// TIA Portal project "Tetsi" (V15.1)

(* hardware
DEVICE "S71500/ET200MP station_1"  S7-1500 station
   slot 0: "Rail_0"  Rack  6ES7 590-1***0-0AA0
   slot 1: "PLC_1"  CPU 1511-1 PN  6ES7 511-1AK02-0AB0  V2.6
      slot 3: "CPU display_1"  6ES7591-1AA00-0AA0
   slot 2: "DI 16x24VDC / DQ 16x24VDC/0.5A BA_1"  DI 16/DQ 16x24VDC  6ES7 523-1BL00-0AA0  V1.0
   slot 3: "AI/AQ 4xU/I/RTD/TC / 2xU/I ST_1"  AI/AQ 4xU/I/RTD/TC / 2xU/I ST  6ES7 534-7QE00-0AB0  V1.0
*)

// ===== PLC "PLC_1"  CPU 1511-1 PN =====

VAR_GLOBAL   // PLC tag table "Default tag table"
   "Clock_Byte" AT %MB0 : Byte;
   "Clock_10Hz" AT %M0.0 : Bool;
   "Clock_5Hz" AT %M0.1 : Bool;
   "Clock_2.5Hz" AT %M0.2 : Bool;
   "Clock_2Hz" AT %M0.3 : Bool;
   "Clock_1.25Hz" AT %M0.4 : Bool;
   "Clock_1Hz" AT %M0.5 : Bool;
   "Clock_0.625Hz" AT %M0.6 : Bool;
   "Clock_0.5Hz" AT %M0.7 : Bool;
   "Tag_1" AT %M100.0 : Bool;
   "Tag_2" AT %M100.2 : Bool;
   "Tag_3" AT %M100.3 : Bool;
   "Tag_4" AT %M100.4 : Bool;
END_VAR

VAR_GLOBAL   // PLC tag table "Tagit"
   "ColorSensor" AT %MW10 : Int;
   "ConveyorEntry" AT %Q0.0 : Bool;
   "ConveyorExit" AT %Q0.1 : Bool;
   "RotationArm" AT %Q0.2 : Bool;
   "RotationArm2" AT %Q0.3 : Bool;
   "RotationArm3" AT %Q0.4 : Bool;
   "StartButton" AT %M12.0 : Bool;
   "StopButton" AT %M12.1 : Bool;
   "ActButton" AT %M12.2 : Bool;
   "RetroreflectiveSensors" AT %M12.3 : Bool;
   "RetroreflectiveSensors2" AT %M12.4 : Bool;
   "RetroreflectiveSensors3" AT %M12.5 : Bool;
END_VAR

DATA_BLOCK "DB"   // DB1
{ S7_Optimized_Access := 'FALSE' }
VERSION : 0.1
   VAR
      nLaatikoita : Int;
      nLaatikoitaSisaan : Int;
      nLaatikoitaUlos : Int;
      kulj2_tyhjenna : Bool;
      kulj1_seis : Bool;
   END_VAR
BEGIN
END_DATA_BLOCK

DATA_BLOCK "Data_block_1"   // DB2
{ S7_Optimized_Access := 'FALSE' }
VERSION : 0.1
   VAR
      start : Bool;
      stop : Bool;
      anturi1 : Bool;
      turvakytkin : Bool;
   END_VAR
BEGIN
END_DATA_BLOCK

DATA_BLOCK "opc_test"   // DB3
{ S7_Optimized_Access := 'TRUE' }
VERSION : 0.1
   VAR
      "bool" : Bool;
      "int" : Int;
   END_VAR
BEGIN
END_DATA_BLOCK

ORGANIZATION_BLOCK "Main"   // OB1, LAD, ProgramCycle
TITLE = "Main Program Sweep (Cycle)"
{ S7_Optimized_Access := 'TRUE' }
VERSION : 0.1
   VAR_INPUT
      Initial_Call : Bool;   // Initial call of this OB
      Remanence : Bool;   // =True, if remanent data are available
   END_VAR
   VAR_TEMP   // added for the SCL form of the ladder/FBD networks
      _w1 : Bool;
      _w2 : Bool;
   END_VAR
BEGIN

REGION Network 1: start/stop
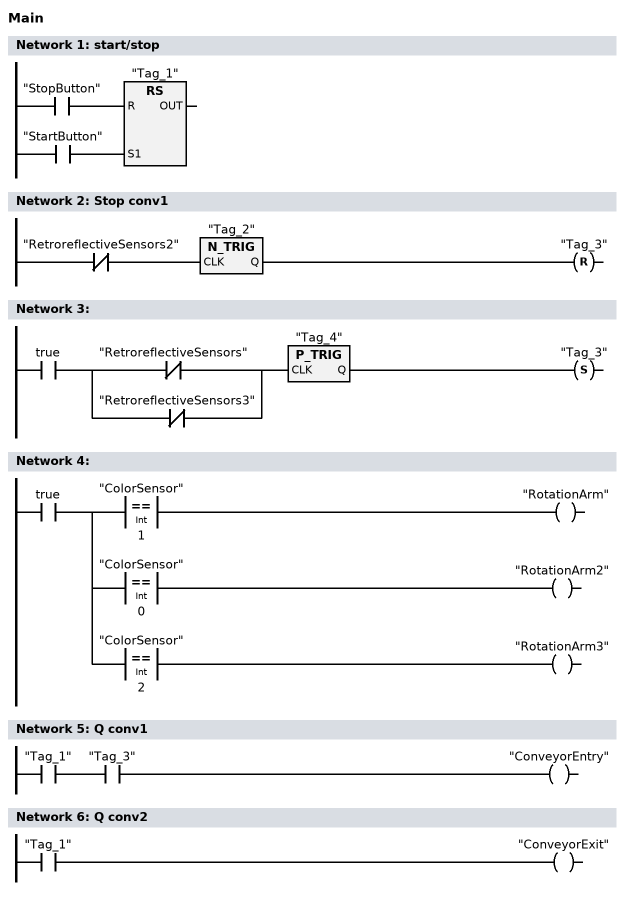
   RUNG wire#powerrail
      Contact( "StopButton" )
      S_RS(operand := "Tag_1", s1 := wire#w1)
   END_RUNG
   RUNG wire#powerrail
      Contact( "StartButton" )
   END_RUNG wire#w1
   // the same network as SCL:
   IF "StopButton" THEN
       "Tag_1" := FALSE;   // RS flip-flop
   END_IF;
   IF "StartButton" THEN "Tag_1" := TRUE; END_IF;
END_REGION

REGION Network 2: Stop conv1
   RUNG wire#powerrail
      I_Contact( "RetroreflectiveSensors2" )
      N_Trig( "Tag_2" )
      R_Coil( "Tag_3" )
   END_RUNG
   // the same network as SCL:
   #_w1 := NOT (NOT "RetroreflectiveSensors2") AND "Tag_2";   // falling edge
   "Tag_2" := NOT "RetroreflectiveSensors2";
   IF #_w1 THEN "Tag_3" := FALSE; END_IF;
END_REGION

REGION Network 3
   RUNG wire#powerrail
      Contact( true )
      wire#w1
      I_Contact( "RetroreflectiveSensors" )
      wire#w2
      P_Trig( "Tag_4" )
      S_Coil( "Tag_3" )
   END_RUNG
   RUNG wire#w1
      I_Contact( "RetroreflectiveSensors3" )
   END_RUNG wire#w2
   // the same network as SCL:
   #_w1 := true AND (NOT "RetroreflectiveSensors" OR NOT "RetroreflectiveSensors3");
   #_w2 := #_w1 AND NOT "Tag_4";   // rising edge
   "Tag_4" := #_w1;
   IF #_w2 THEN "Tag_3" := TRUE; END_IF;
END_REGION

REGION Network 4
   RUNG wire#powerrail
      Contact( true )
      wire#w1
      { S7_Templates := "SrcType := Int" } EQ_Contact(in1 := "ColorSensor", in2 := 1)
      Coil( "RotationArm" )
   END_RUNG
   RUNG wire#w1
      { S7_Templates := "SrcType := Int" } EQ_Contact(in1 := "ColorSensor", in2 := 0)
      Coil( "RotationArm2" )
   END_RUNG
   RUNG wire#w1
      { S7_Templates := "SrcType := Int" } EQ_Contact(in1 := "ColorSensor", in2 := 2)
      Coil( "RotationArm3" )
   END_RUNG
   // the same network as SCL:
   "RotationArm" := true AND ("ColorSensor" = 1);
   "RotationArm2" := true AND ("ColorSensor" = 0);
   "RotationArm3" := true AND ("ColorSensor" = 2);
END_REGION

REGION Network 5: Q conv1
   RUNG wire#powerrail
      Contact( "Tag_1" )
      Contact( "Tag_3" )
      Coil( "ConveyorEntry" )
   END_RUNG
   // the same network as SCL:
   "ConveyorEntry" := "Tag_1" AND "Tag_3";
END_REGION

REGION Network 6: Q conv2
   RUNG wire#powerrail
      Contact( "Tag_1" )
      Coil( "ConveyorExit" )
   END_RUNG
   // the same network as SCL:
   "ConveyorExit" := "Tag_1";
END_REGION
END_ORGANIZATION_BLOCK